FUNCTION_BLOCK PICKER_HMI_ADP (* Composite FB For HMI Plug *)
  (* Standard: 61499-2 *)
  (* Version 0.2, 2003-12-05, JHC, Rockwell Automation, Renamed from NEWCOMPFB. *)
  (* Version 0.1, 2002-01-08, JHC, Rockwell Automation, Added DLY FB as example. *)
  (* Version 0.0, 2000-05-27, JHC, Rockwell Automation *)
  (* Compiler header: package fb.rt.pnp; *)
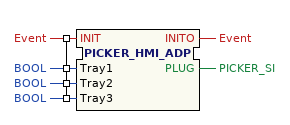
  EVENT_INPUT
    INIT WITH Tray1, Tray2, Tray3; (* Initialization Request *)
  END_EVENT
  EVENT_OUTPUT
    INITO; (* Initialization Confirm *)
  END_EVENT
  VAR_INPUT
    Tray1 : BOOL;
    Tray2 : BOOL;
    Tray3 : BOOL;
  END_VAR
  PLUGS
    PLUG : PICKER_SI;
  END_PLUGS
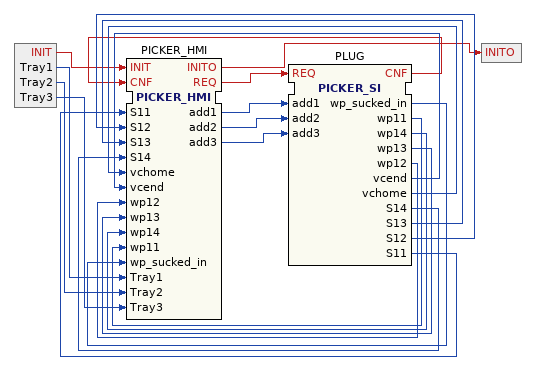
  FBS
    PICKER_HMI : PICKER_HMI;
  END_FBS
  EVENT_CONNECTIONS
    INIT TO PICKER_HMI.INIT;
    PICKER_HMI.INITO TO INITO;
    PICKER_HMI.REQ TO PLUG.REQ;
    PLUG.CNF TO PICKER_HMI.CNF;
  END_CONNECTIONS
  DATA_CONNECTIONS
    PLUG.wp_sucked_in TO PICKER_HMI.wp_sucked_in;
    PLUG.wp11 TO PICKER_HMI.wp11;
    PLUG.wp14 TO PICKER_HMI.wp14;
    PLUG.wp13 TO PICKER_HMI.wp13;
    PLUG.wp12 TO PICKER_HMI.wp12;
    PLUG.vcend TO PICKER_HMI.vcend;
    PLUG.vchome TO PICKER_HMI.vchome;
    PLUG.S14 TO PICKER_HMI.S14;
    PLUG.S13 TO PICKER_HMI.S13;
    PLUG.S12 TO PICKER_HMI.S12;
    PLUG.S11 TO PICKER_HMI.S11;
    PICKER_HMI.add1 TO PLUG.add1;
    PICKER_HMI.add2 TO PLUG.add2;
    PICKER_HMI.add3 TO PLUG.add3;
    Tray1 TO PICKER_HMI.Tray1;
    Tray2 TO PICKER_HMI.Tray2;
    Tray3 TO PICKER_HMI.Tray3;
  END_CONNECTIONS
END_FUNCTION_BLOCK
